// TIA Portal project "Lab_3" (V15.1)

(* hardware
DEVICE "ET 200SP station_1"  ET 200SP-Station
   slot 0: "Rack_0"  Rack  6ES5 710-8MAx1
   slot 1: "PLC_1"  CPU 1512SP F-1 PN  6ES7 512-1SK01-0AB0  V2.6
   slot 2: "DI 8x24VDC HF_1"  DI 8x24VDC HF  6ES7 131-6BF00-0CA0  V2.0
      slot 1: "DI 8x24VDC HF_1"  DI 8x24VDC HF
   slot 3: "DI 8x24VDC HF_2"  DI 8x24VDC HF  6ES7 131-6BF00-0CA0  V2.0
      slot 1: "DI 8x24VDC HF_2"  DI 8x24VDC HF
   slot 4: "DQ 8x24VDC/0.5A HF_1"  DQ 8x24VDC/0.5A HF  6ES7 132-6BF00-0CA0  V2.0
      slot 1: "DQ 8x24VDC/0.5A HF_1"  DQ 8x24VDC/0.5A HF
   slot 5: "DQ 8x24VDC/0.5A HF_2"  DQ 8x24VDC/0.5A HF  6ES7 132-6BF00-0CA0  V2.0
      slot 1: "DQ 8x24VDC/0.5A HF_2"  DQ 8x24VDC/0.5A HF
   slot 6: "CM 4xIO-Link_1"  CM 4xIO-Link  6ES7 137-6BD00-0BA0  V2.2
      slot 1: "CM 4xIO-Link_1"  6ES7 137-6BD00-0BA0
   slot 7: "Server module_1"  Server module  6ES7 193-6PA00-0AA0  V1.1
      slot 1: "Server module_1"  Server module
   slot 127: "BA 2xRJ45"  BA 2xRJ45  6ES7 193-6AR00-0AA0  V0.0
      slot 32769: "Port_1"  6ES7 193-6AR00-0AA0
      slot 32770: "Port_2"  6ES7 193-6AR00-0AA0
*)

// ===== PLC "PLC_1"  CPU 1512SP F-1 PN =====

VAR_GLOBAL   // PLC tag table "CP-L-Conveyor"
   "start_btn" AT %I1.0 : Bool;   // True = Start button pushed
   "stop_btn" AT %I1.1 : Bool;   // False = Stop button pushed
   "op-mode_btn" AT %I1.2 : Bool;   // Select operation mode (False = Setup mode, True = Automatic mode)
   "reset_btn" AT %I1.3 : Bool;   // True = Reset button pushed
   "carrier_stopper_pos" AT %I1.4 : Bool;   // True = Carrier detected at stopper position (corresponds to ident code bit 0)
   "emergency_stop_btn" AT %I1.5 : Bool;   // False = Emergency stop button pushed (n.c.)
   "carrier_entry_pos" AT %I1.6 : Bool;   // True = Carrier detected at conveyor entry
   "carrier_exit_pos" AT %I1.7 : Bool;   // True = Carrier detected at conveyor exit
   "carrier_ident_0" AT %I42.0 : Bool;   // True = Carrier ident code bit 0 detected
   "carrier_ident_1" AT %I42.1 : Bool;   // True = Carrier ident code bit 1 detected
   "carrier_ident_2" AT %I42.2 : Bool;   // True = Carrier ident code bit 2 detected
   "carrier_ident_3" AT %I42.3 : Bool;   // True = Carrier ident code bit 3 detected
   "switch_S1" AT %I42.4 : Bool;   // A = True = Encoder A signal detcted, R = False = Coupling signal right detected
   "switch_S2" AT %I42.5 : Bool;   // B = True = Encoder B signal detected, L = False = Coupling signal left detected
   "stop_cylinder_low_pos" AT %I42.7 : Bool;   // True = Stopper cylinder in lower end position
   "start_btn_light" AT %Q1.0 : Bool;   // True = Switch on start button signal light
   "reset_btn_light" AT %Q1.1 : Bool;   // True = Switch on reset button signal light
   "func_Q1_light" AT %Q1.2 : Bool;   // True = Switch on special function Q1 signal light
   "func_Q2_light" AT %Q1.3 : Bool;   // True = Switch on special function Q2 signal light
   "belt_forward" AT %Q1.4 : Bool;   // True = Drive belt in forward direction
   "belt_reverse" AT %Q1.5 : Bool;   // True = Drive belt in reverse direction
   "belt_speed" AT %Q1.6 : Bool;   // Select belt speed (False = normal, True = slow)
   "move_cylinder_down" AT %Q1.7 : Bool;   // True = Move stopper cylinder down
   "coupling_signal_left" AT %Q42.4 : Bool;   // True = Send coupling signal left
   "coupling_signal_right" AT %Q42.5 : Bool;   // True = Send coupling signal right
END_VAR

DATA_BLOCK "CP-L-Conveyor_DB"   // DB2
{ S7_Optimized_Access := 'TRUE' }
VERSION : 0.1
// stored: InstanceOfName CP-L-Conveyor
"CP-L-Conveyor"
BEGIN
END_DATA_BLOCK

// folder: System blocks/Program resources

DATA_BLOCK "IEC_Timer_0_DB"   // DB1
{ S7_Optimized_Access := 'TRUE' }
AUTHOR : Simatic
FAMILY : IEC
NAME : IEC_TMR
VERSION : 1.0
// stored: InstanceOfName IEC_TIMER
"IEC_TIMER"
BEGIN
END_DATA_BLOCK

// folder: (top level)

FUNCTION_BLOCK "CP-L-Conveyor"   // FB1, SCL
{ S7_Optimized_Access := 'TRUE' }
VERSION : 0.1
   VAR_INPUT
      Xstartbtn : Bool;
      Xstopbtn : Bool;
      "Xop-mode_btn" : Bool;
      Xreset_btn : Bool;
      Xcarrier_stopper_pos : Bool;
      Xemergency_stop_btn : Bool;
      Xcarrier_entry_pos : Bool;
      Xcarrier_exit_pos : Bool;
      Xcarrier_ident_0 : Bool;
      Xcarrier_ident_1 : Bool;
      Xcarrier_ident_2 : Bool;
      Xcarrier_ident_3 : Bool;
      Xswitch_S1 : Bool;
      Xswitch_S2 : Bool;
      Xstop_cylinder_low_pos : Bool;
   END_VAR
   VAR_OUTPUT
      Ystart_btn_light : Bool := false;
      Y_reset_btn_light : Bool := false;
      Yfunc_Q1_light : Bool;
      Yfunc_Q2_light : Bool;
      Ybelt_forward : Bool;
      Ybelt_reverse : Bool;
      Ybelt_speed : Bool;
      Ymove_cylinder_down : Bool;
      Ycoupling_signal_left : Bool;
      Ycoupling_signal_right : Bool;
   END_VAR
BEGIN
   IF #"Xop-mode_btn" = TRUE THEN
       IF #Xcarrier_entry_pos = TRUE THEN
           #Ybelt_forward := TRUE;
       END_IF;
       IF #Xcarrier_exit_pos = TRUE THEN
           #Ybelt_forward := FALSE;
       END_IF;
   //ELSE
   END_IF;
   "IEC_Timer_0_DB".TON(IN:=#Xcarrier_stopper_pos,
                        PT:=T#3S,
                        Q=>#Ymove_cylinder_down);
END_FUNCTION_BLOCK

ORGANIZATION_BLOCK "Main"   // OB1, SCL, ProgramCycle
TITLE = "Main Program Sweep (Cycle)"
{ S7_Optimized_Access := 'TRUE' }
VERSION : 0.1
   VAR_INPUT
      Initial_Call : Bool;   // Initial call of this OB
      Remanence : Bool;   // =True, if remanent data are available
   END_VAR
BEGIN
   "CP-L-Conveyor_DB"(Xstartbtn:="start_btn",
                      Xstopbtn:="stop_btn",
                      "Xop-mode_btn":="op-mode_btn",
                      Xreset_btn:="reset_btn",
                      Xcarrier_stopper_pos:="carrier_stopper_pos",
                      Xemergency_stop_btn:="emergency_stop_btn",
                      Xcarrier_entry_pos:="carrier_entry_pos",
                      Xcarrier_exit_pos:="carrier_exit_pos",
                      Xcarrier_ident_0:="carrier_ident_0",
                      Xcarrier_ident_1:="carrier_ident_1",
                      Xcarrier_ident_2:="carrier_ident_2",
                      Xcarrier_ident_3:="carrier_ident_3",
                      Xswitch_S1:="switch_S1",
                      Xswitch_S2:="switch_S2",
                      Xstop_cylinder_low_pos:="stop_cylinder_low_pos",
                      Ystart_btn_light=>"start_btn_light",
                      Y_reset_btn_light=>"reset_btn_light",
                      Yfunc_Q1_light=>"func_Q1_light",
                      Yfunc_Q2_light=>"func_Q2_light",
                      Ybelt_forward=>"belt_forward",
                      Ybelt_reverse=>"belt_reverse",
                      Ybelt_speed=>"belt_speed",
                      Ymove_cylinder_down=>"move_cylinder_down",
                      Ycoupling_signal_left=>"coupling_signal_left",
                      Ycoupling_signal_right=>"coupling_signal_right");
END_ORGANIZATION_BLOCK